% RSLogix 500 project dimag laga bhai.RSS, saved by version 8.30.00.15 %
PROJECT "UNTITLED"    % processor: MicroLogix 1000 %

PROGRAM FILES
  LAD 2 "MAIN_PROG"  7 rungs
  LAD 3 "USER_FAULT"  1 rungs
  LAD 4 "HSC_INT"  1 rungs
  LAD 5 "STI_INT"  1 rungs
  LAD 6, 7, 8, 9, 10, 11, 12, 13, 14, 15, 16: only END

DATA FILES
  O0 OUTPUT  1 elements
  I1 INPUT  2 elements
  S2 STATUS  33 elements
  B3 BINARY  32 elements
  T4 TIMER  40 elements
  C5 COUNTER  32 elements
  R6 CONTROL  16 elements
  N7 INTEGER  105 elements

LADDER 2 "MAIN_PROG"
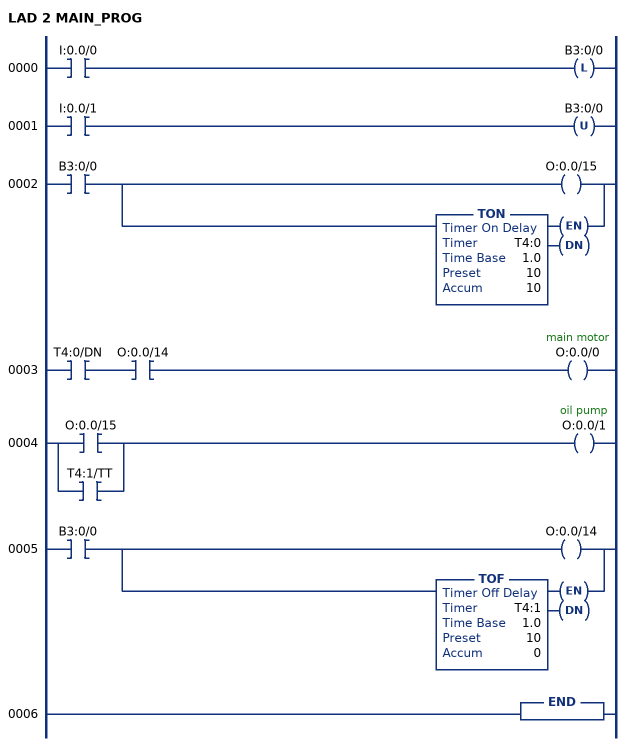
% Rung: 0 %
SOR XIC I:0.0/0 OTL B3:0/0 EOR
% Rung: 1 %
SOR XIC I:0.0/1 OTU B3:0/0 EOR
% Rung: 2 %
SOR XIC B3:0/0 BST OTE O:0.0/15 NXB TON T4:0 1.0 10 10 BND EOR
% Rung: 3 %
SOR XIC T4:0/DN XIC O:0.0/14 OTE O:0.0/0 EOR
%   O:0.0/0  "main motor" %
% Rung: 4 %
SOR BST XIC O:0.0/15 NXB XIC T4:1/TT BND OTE O:0.0/1 EOR
%   O:0.0/1  "oil pump" %
% Rung: 5 %
SOR XIC B3:0/0 BST OTE O:0.0/14 NXB TOF T4:1 1.0 10 0 BND EOR
% Rung: 6 %
SOR END EOR

DATA TABLE (non-zero values as saved)
DATA T4
% .PRE .ACC %
% T4:0 % 10 10
% T4:1 % 10 0
